// TwinCAT 3 PLC project PLC1
// ProgramVersion: 3.1.4023.0
// libraries:
//   Tc2_Standard, * (Beckhoff Automation GmbH)
//   Tc2_System, * (Beckhoff Automation GmbH)
//   Tc3_Module, * (Beckhoff Automation GmbH)
// project tree:
//   GVLs/ GVL.TcGVL
//   / PlcTask.TcTTO
//   POUs/ MAIN.TcPOU
// real-time tasks:
//   TASK PlcTask1: cycle T#250us, priority 21, ADS port 350
// I/O:
//   DEVICE Device 3 (EtherCAT), AmsNetId 192.168.56.1.4.1
//     Box 1 (Q.station 101 T) [Q.station 101 T]
//     Box 2 (lan9252) [lan9252]

CONFIGURATION PLC1
    RESOURCE PLC ON TwinCAT3
        TASK PlcTask(INTERVAL := T#250us, PRIORITY := 21);
        PROGRAM MAIN WITH PlcTask : MAIN;
    END_RESOURCE
END_CONFIGURATION

// ---- GVLs/GVL.TcGVL
{attribute 'qualified_only'}
VAR_GLOBAL
	DI1X AT %I*: USINT;
	DI2X AT %I*: USINT;
END_VAR

// ---- POUs/MAIN.TcPOU
PROGRAM MAIN
VAR
	DI2 AT %I*: USINT;
	DI1 AT %I*: USINT;
END_VAR
VAR_OUTPUT
	OUTDI2: USINT;
	OUTDI1: USINT;
END_VAR
VAR
	Count AT %I*: REAL;
END_VAR
VAR_OUTPUT
	Count_Out: REAL;
END_VAR

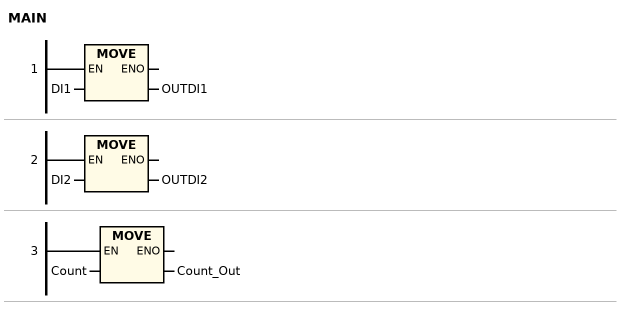
// NETWORK 1
OUTDI1 := DI1;

// NETWORK 2
OUTDI2 := DI2;

// NETWORK 3
Count_Out := Count;

END_PROGRAM
